{attribute 'strict'}
TYPE E_CognexCameraGetFileStatus :
(
	WAITING_FOR_STATUS_CODE						:= 2,
	THE_COMMAND_WAS_EXECUTED_SUCCESSFULLY		:= 1,
	UNRECOGNIZED_COMMAND 						:= 0,
	THE_ACTIVE_JOB_HAS_NOT_BEEN_SAVED 			:= -2
);
END_TYPE

(* stored: Version 1.1.0.1, ProductVersion 3.1.4024.9
   DUT E_CognexCameraGetFileStatus: Id {2cea9dfc-3f2a-4d3d-a217-95cf1573239b} *)
